Yaskawa INFORM job: ARGPASS.JBI

/JOB
//NAME ARGPASS
//POS
///NPOS 0,0,0,0,0,0
//INST
///DATE 2026/05/07 11:26
///ATTR SC,RW
///GROUP1 RB1
NOP
'PASS THRU ENTRYPOINT:
'ARGF5 FROM CALLER IS FORWARDED TO TOOLCHANGE_V2 AS ARG#1
'USE THIS WHEN EXTERNAL LOGIC/HMI WRITES REQUEST TO ARGF5
CALL JOB:TOOLCHANGE_V2 ARGF5
END
